(* PLC project Unnamed, Unknown Unnamed 1 *)
(* stored: creationDateTime 2026-05-01T18:15:01, modificationDateTime 2026-05-01T20:57:57 *)

PROGRAM program0Project_02_Tank_Level
  VAR
    PB_EStop AT %IX0.0 : BOOL;
    PB_FaultReset AT %IX0.1 : BOOL;
    SW_ModeAuto AT %IX0.2 : BOOL;
    LS_LowLow AT %IX0.3 : BOOL;
    LS_Low AT %IX0.4 : BOOL;
    LS_High AT %IX0.5 : BOOL;
    LS_HighHigh AT %IX0.6 : BOOL;
    PB_ManDrain AT %IX0.7 : BOOL;
    MP1_FillPump AT %QX0.0 : BOOL;
    SV1_FillValve AT %QX0.1 : BOOL;
    SV2_DrainValve AT %QX0.2 : BOOL;
    HL1_RunLamp AT %QX0.3 : BOOL;
    HL2_AlarmLamp AT %QX0.4 : BOOL;
    HL3_DrainLamp AT %QX0.5 : BOOL;
    MR_MasterEnable AT %MX0.0 : BOOL;
    MR_FaultOverflow AT %MX0.1 : BOOL;
    MR_FaultDryRun AT %MX0.2 : BOOL;
    MR_FaultAny AT %MX0.3 : BOOL;
    MR_AutoMode AT %MX0.4 : BOOL;
    MR_ManualMode AT %MX0.5 : BOOL;
    MR_FillActive AT %MX0.6 : BOOL;
    MR_DrainActive AT %MX0.7 : BOOL;
    MR_TankEmpty AT %MX1.0 : BOOL;
    MR_TankFull AT %MX1.1 : BOOL;
    MR_FaultFillTimeout AT %MX1.2 : BOOL;
    MR_FaultDrainTimeout AT %MX1.3 : BOOL;
  END_VAR
  VAR
    Clock_1Hz : BOOL;
    TON_DryRunDelay : TON;
    DryRunTime : TIME := T#5s;
    FillTimeoutTime : TIME := T#120s;
    DrainTimeoutTime : TIME := T#180s;
    TON_FillTimeout : TON;
  END_VAR

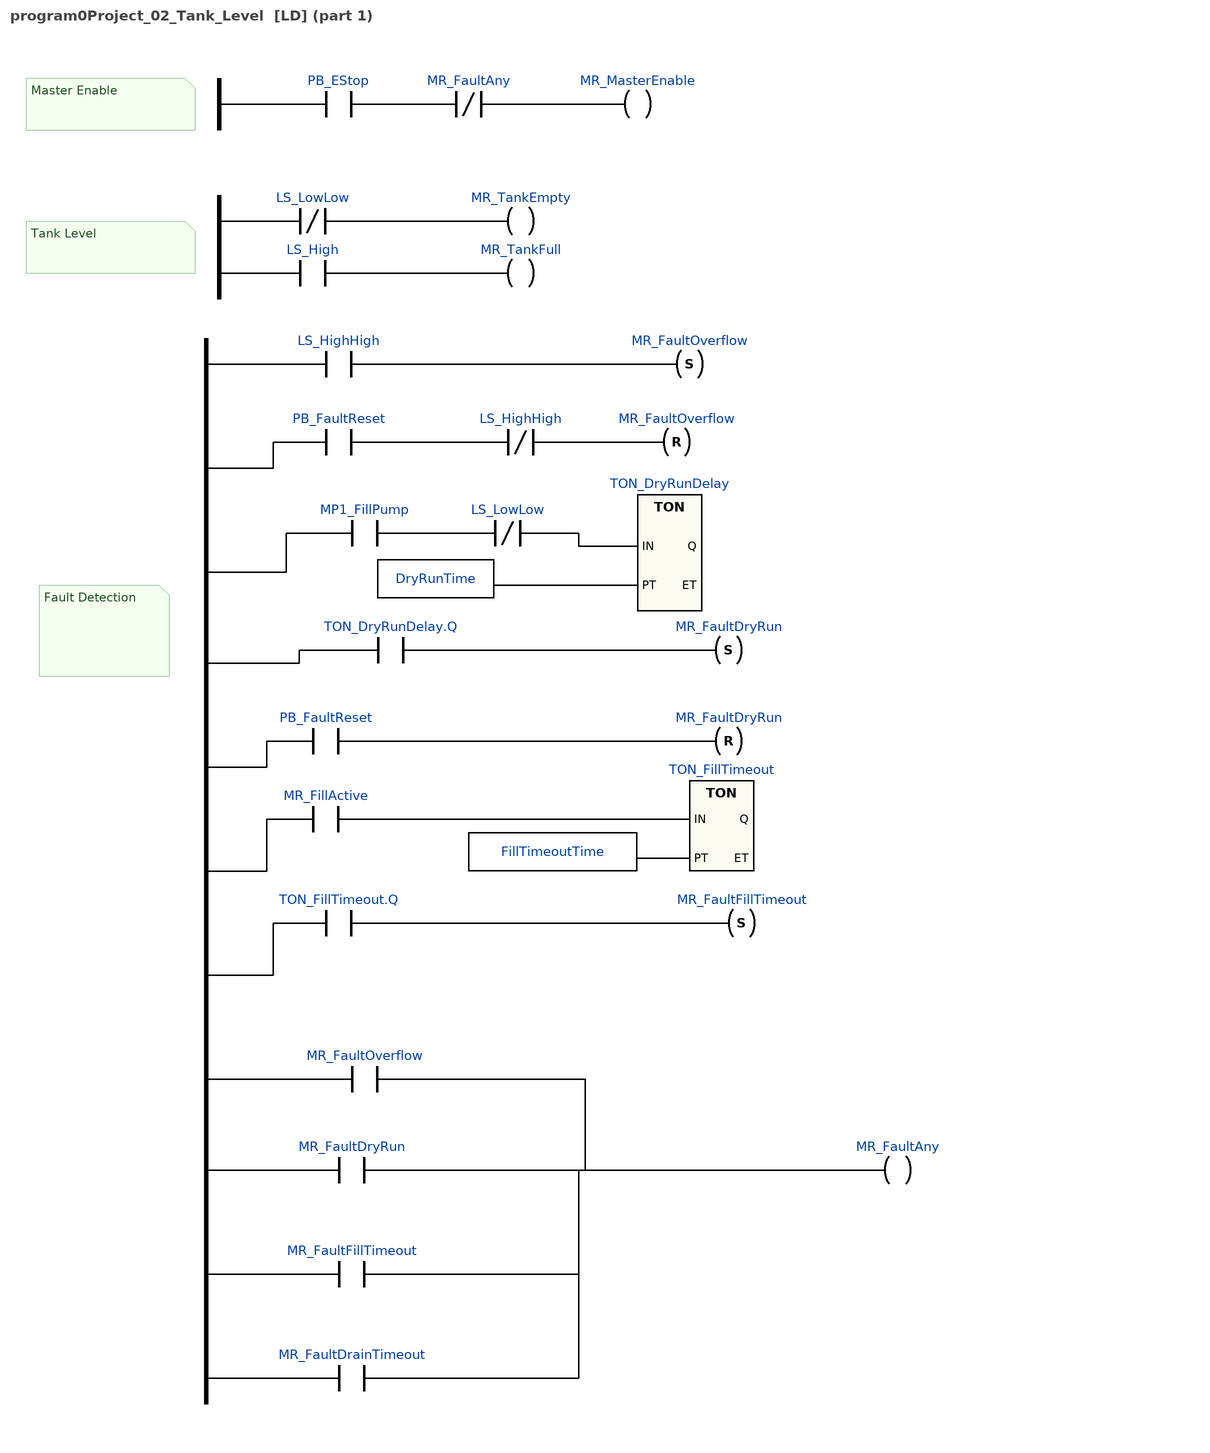
(* LD diagram, written out as Structured Text *)
(* Master Enable *)
MR_MasterEnable := PB_EStop AND NOT MR_FaultAny;
MR_TankEmpty := NOT LS_LowLow;
(* Tank Level *)
MR_TankFull := LS_High;
IF LS_HighHigh THEN MR_FaultOverflow := TRUE; END_IF;
IF PB_FaultReset AND NOT LS_HighHigh THEN MR_FaultOverflow := FALSE; END_IF;
(* Fault Detection *)
IF TON_DryRunDelay.Q THEN MR_FaultDryRun := TRUE; END_IF;
IF PB_FaultReset THEN MR_FaultDryRun := FALSE; END_IF;
IF TON_FillTimeout.Q THEN MR_FaultFillTimeout := TRUE; END_IF;
MR_FaultAny := MR_FaultDryRun OR MR_FaultOverflow OR MR_FaultFillTimeout OR MR_FaultDrainTimeout;
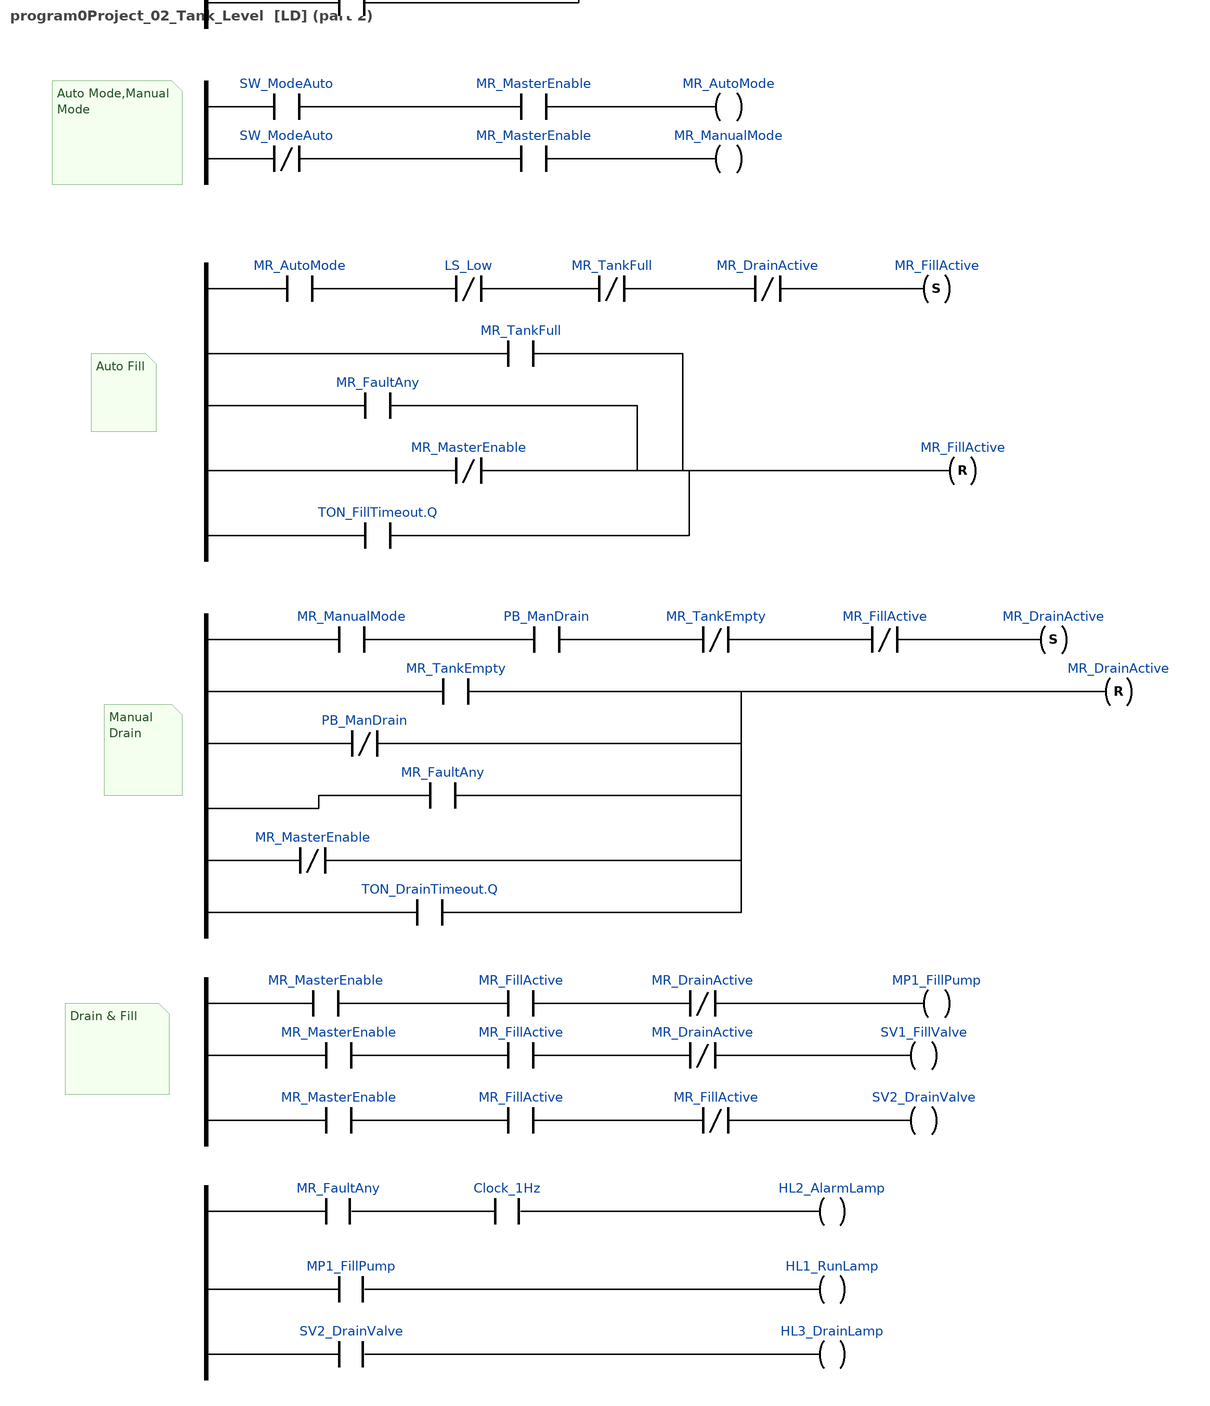
(* Auto Mode,Manual Mode *)
MR_AutoMode := SW_ModeAuto AND MR_MasterEnable;
MR_ManualMode := NOT SW_ModeAuto AND MR_MasterEnable;
IF MR_AutoMode AND NOT LS_Low AND NOT MR_TankFull AND NOT MR_DrainActive THEN MR_FillActive := TRUE; END_IF;
(* Auto Fill *)
IF NOT MR_MasterEnable OR TON_FillTimeout.Q OR MR_FaultAny OR MR_TankFull THEN MR_FillActive := FALSE; END_IF;
IF MR_ManualMode AND PB_ManDrain AND NOT MR_TankEmpty AND NOT MR_FillActive THEN MR_DrainActive := TRUE; END_IF;
IF MR_TankEmpty OR NOT PB_ManDrain OR MR_FaultAny OR NOT MR_MasterEnable OR TON_DrainTimeout.Q THEN MR_DrainActive := FALSE; END_IF;
(* Manual Drain *)
MP1_FillPump := MR_MasterEnable AND MR_FillActive AND NOT MR_DrainActive;
(* Drain & Fill *)
SV1_FillValve := MR_MasterEnable AND MR_FillActive AND NOT MR_DrainActive;
SV2_DrainValve := MR_MasterEnable AND MR_FillActive AND NOT MR_FillActive;
HL2_AlarmLamp := MR_FaultAny AND Clock_1Hz;
HL1_RunLamp := MP1_FillPump;
HL3_DrainLamp := SV2_DrainValve;
TON_DryRunDelay(IN := MP1_FillPump AND NOT LS_LowLow, PT := DryRunTime);
TON_FillTimeout(IN := MR_FillActive, PT := FillTimeoutTime);
END_PROGRAM

CONFIGURATION Config0
  RESOURCE Res0 ON PLC
    TASK task0(INTERVAL := T#20ms, PRIORITY := 0);
    PROGRAM instance0 WITH task0 : program0Project_02_Tank_Level;
  END_RESOURCE
END_CONFIGURATION
